// SIMATIC S7-200 SMART project (STEP 7-Micro/WIN SMART), CPU ST20

SYMBOL_TABLE Table 1
CON_Done         M0.0
CON_Busy         M0.1
CON_Error        M0.2
CON_Stat         MB1
RECV_Done        M2.0
RECV_Busy        M2.1
RECV_Error       M2.2
RECV_Stat        MB3
RECV_Len         MW4
END_SYMBOL_TABLE

SYMBOL_TABLE System Symbols
Always_On        SM0.0    // Always ON
First_Scan_On    SM0.1    // ON for the first scan cycle only
END_SYMBOL_TABLE

ORGANIZATION_BLOCK MAIN:OB1
TITLE=Program Comments
BEGIN
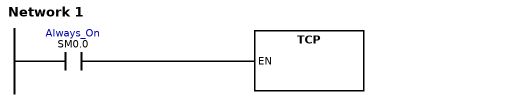
Network 1
LD     Always_On:SM0.0
CALL   TCP:SBR12
END_ORGANIZATION_BLOCK

// SBR10: protected block, not included

// SBR11: protected block, not included

SUBROUTINE_BLOCK TCP:SBR12
TITLE=Subroutine Comments
BEGIN
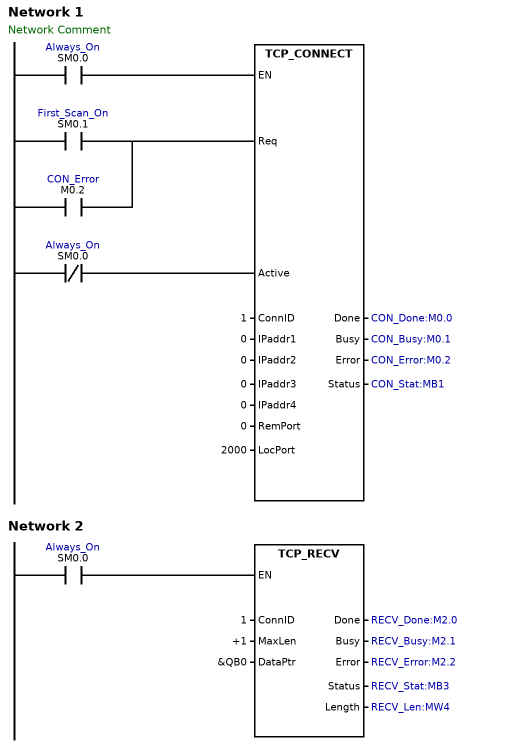
Network 1
// Network Comment
LD     Always_On:SM0.0
=      L60.0
LD     First_Scan_On:SM0.1
O      CON_Error:M0.2
=      L63.7
LDN    Always_On:SM0.0
=      L63.6
LD     L60.0
CALL   TCP_CONNECT:SBR10, L63.7, L63.6, 1, 0, 0, 0, 0, 0, 2000, CON_Done:M0.0, CON_Busy:M0.1, CON_Error:M0.2, CON_Stat:MB1
Network 2
// (network saved uncompiled; LAD cells follow)
// row 0: c0 -| |- Always_On:SM0.0  c1 --  c2 [TCP_RECV EN:=power@row0, ConnID:=1, MaxLen:=+1, DataPtr:=&QB0, Done=>RECV_Done:M2.0, Busy=>RECV_Busy:M2.1, Error=>RECV_Error:M2.2, Status=>RECV_Stat:MB3, Length=>RECV_Len:MW4]
// row 1: c2 [box]
// row 2: c2 [box]
END_SUBROUTINE_BLOCK
